// TIA Portal V17 export
// export: Created 2025-08-05T09:36:02.3274089Z, ExportSetting WithDefaults, DisplayName Totally Integrated Automation Portal, DisplayVersion V17, DisplayName TIA Portal Openness, DisplayVersion V17, DisplayName TIA Portal Version Control Interface, DisplayVersion V17, DisplayName SINAMICS Startdrive Advanced, DisplayVersion V17, DisplayName SINAMICS Startdrive G130, G150, S120, S150, SINAMICS MV, S210, DisplayVersion V17, DisplayName SINAMICS Startdrive G110M, G120, G120C, G120D, G120P, G115D, DisplayVersion V17, DisplayName STEP 7 Professional, DisplayVersion V17, DisplayName STEP 7 Safety, DisplayVersion V17, DisplayName WinCC Advanced, DisplayVersion V17
TYPE "typeSmcChillerHrle90a40cmIo"
// stored: IsFailsafeCompliant false
   STRUCT
      in { ExternalAccessible := 'False'; ExternalVisible := 'False'; ExternalWritable := 'False'} : Struct   // Lesen / Read
         fluidDischargeTempCH1 { ExternalAccessible := 'False'; ExternalVisible := 'False'; ExternalWritable := 'False'} : Real;   // Austrittstemperatur der zirkulierenden Flüssigkeit Kanal 1 / Outlet temperature of the circulating fluid channel 1
         fluidDischargeTempCH2 { ExternalAccessible := 'False'; ExternalVisible := 'False'; ExternalWritable := 'False'} : Real;   // Austrittstemperatur der zirkulierenden Flüssigkeit Kanal 2 / Outlet temperature of the circulating fluid channel 2
         reserve1 { ExternalAccessible := 'False'; ExternalVisible := 'False'; ExternalWritable := 'False'} : Word;   // Reserve
         reserve2 { ExternalAccessible := 'False'; ExternalVisible := 'False'; ExternalWritable := 'False'} : Word;   // Reserve
         fluidDischargePressureCH1 { ExternalAccessible := 'False'; ExternalVisible := 'False'; ExternalWritable := 'False'} : Real;   // Förderdruck der zirkulierenden Flüssigkeit Kanal 1 / Delivery pressure of the circulating fluid channel 1
         reserve3 { ExternalAccessible := 'False'; ExternalVisible := 'False'; ExternalWritable := 'False'} : Word;   // Reserve
         reserve4 { ExternalAccessible := 'False'; ExternalVisible := 'False'; ExternalWritable := 'False'} : Word;   // Reserve
         reserve5 { ExternalAccessible := 'False'; ExternalVisible := 'False'; ExternalWritable := 'False'} : Word;   // Reserve
         dataDisplay1 { ExternalAccessible := 'False'; ExternalVisible := 'False'; ExternalWritable := 'False'} : Real;   // Datenanzeige 1 / Data display 1
         dataDisplay2 { ExternalAccessible := 'False'; ExternalVisible := 'False'; ExternalWritable := 'False'} : Real;   // Datenanzeige 2 / Data display 2
         statusFlags1 { ExternalAccessible := 'False'; ExternalVisible := 'False'; ExternalWritable := 'False'} : Array[0..15] of Bool;   // Statuskennzeichen 1 / Status identifier 1
         alarmFlags1 { ExternalAccessible := 'False'; ExternalVisible := 'False'; ExternalWritable := 'False'} : Array[0..15] of Bool;   // Alarmmerker 1 / Alarm flag 1
         alarmFlags2 { ExternalAccessible := 'False'; ExternalVisible := 'False'; ExternalWritable := 'False'} : Array[0..15] of Bool;   // Alarmmerker 2 / Alarm flag 2
         alarmFlags3 { ExternalAccessible := 'False'; ExternalVisible := 'False'; ExternalWritable := 'False'} : Array[0..15] of Bool;   // Alarmmerker 3 / Alarm flag 3
         alarmFlags4 { ExternalAccessible := 'False'; ExternalVisible := 'False'; ExternalWritable := 'False'} : Array[0..15] of Bool;   // Alarmmerker 4 / Alarm flag 4
         alarmFlags5 { ExternalAccessible := 'False'; ExternalVisible := 'False'; ExternalWritable := 'False'} : Array[0..15] of Bool;   // Alarmmerker 5 / Alarm flag 5
      END_STRUCT;
      inOut { ExternalAccessible := 'False'; ExternalVisible := 'False'; ExternalWritable := 'False'} : Struct   // Lesen/Schreiben / Read/write
         fluidSetTempCH1 { ExternalAccessible := 'False'; ExternalVisible := 'False'; ExternalWritable := 'False'} : Real;   // Solltemperatur der zirkulierenden Flüssigkeit / Target temperature of the circulating fluid
         fluidSetTempCH2 { ExternalAccessible := 'False'; ExternalVisible := 'False'; ExternalWritable := 'False'} : Real;   // Umwälzflüssigkeitssolltemperatur als Offset von Kanal 1 (Sollwert Kanal 2 = Sollwert Kanal 1 + Offset Kanal 2) / Circulating fluid target temperature as offset for channel 1 (target value channel 2 = target value channel 1 + offset channel 2)
         controlBits { ExternalAccessible := 'False'; ExternalVisible := 'False'; ExternalWritable := 'False'} : Array[0..15] of Bool;   // Steuerbits / Control bits
         dataInstr { ExternalAccessible := 'False'; ExternalVisible := 'False'; ExternalWritable := 'False'} : Array[0..1] of Byte;   // Datenanweisungen / Data instructions
      END_STRUCT;
   END_STRUCT;
   // // in.statusFlags1[0] : Laufstatus / Running status
   // // in.statusFlags1[1] : Betriebsstoppalarm ausgelöst Status / Stop operation alarm triggered status
   // // in.statusFlags1[2] : Betriebsfortsetzungsalarm ausgelöst / Continue operation alarm triggered
   // // in.statusFlags1[3] : Reserve
   // // in.statusFlags1[4] : Abschluss der Vorbereitung (TEMP READY) Status / End of preparation (TEMP READY) status
   // // in.statusFlags1[5] : Reserve
   // // in.statusFlags1[6] : Reserve
   // // in.statusFlags1[7] : Reserve
   // // in.statusFlags1[8] : Reserve
   // // in.statusFlags1[9] : Reserve
   // // in.statusFlags1[10] : Reserve
   // // in.statusFlags1[11] : Reserve
   // // in.statusFlags1[12] : Reserve
   // // in.statusFlags1[13] : Reserve
   // // in.statusFlags1[14] : Reserve
   // // in.statusFlags1[15] : Gefrierschutzstatus / Freeze protection status
   // // in.alarmFlags1[0] : Niedriger Flüssigkeitsstand im Tank / Low fluid level in the tank
   // // in.alarmFlags1[1] : CH1 abnorm hohe Temperatur der zirkulierenden Flüssigkeit / CH1 abnormally high temperature of the circulating fluid
   // // in.alarmFlags1[2] : Reserve
   // // in.alarmFlags1[3] : Reserve
   // // in.alarmFlags1[4] : Ungewöhnlich hohe Rücklauftemperatur der zirkulierenden Flüssigkeit / Unusually high return temperature of the circulating fluid
   // // in.alarmFlags1[5] : Ungewöhnlich hoher Auslassdruck der zirkulierenden Flüssigkeit / Unusually high outlet pressure of the circulating fluid
   // // in.alarmFlags1[6] : Reserve
   // // in.alarmFlags1[7] : Hoher Druckanstieg der zirkulierenden Flüssigkeit / High pressure increase of the circulating fluid
   // // in.alarmFlags1[8] : Hoher Druckabfall der zirkulierenden Flüssigkeit / High pressure of the circulating fluid
   // // in.alarmFlags1[9] : Reserve
   // // in.alarmFlags1[10] : Ungewöhnlich niedrige Ansaugtemperatur des Kompressors / Unusually low intake temperature of the compressor
   // // in.alarmFlags1[11] : Reserve
   // // in.alarmFlags1[12] : Unnormaler Anstieg des Drucks im Kältemittelkreislauf (Hochdruckseite) / Abnormal pressure rise in the coolant circuit (high pressure side)
   // // in.alarmFlags1[13] : Reserve
   // // in.alarmFlags1[14] : Kältemittelleck / Coolant leak
   // // in.alarmFlags1[15] : Ungewöhnlicher Anstieg des Drucks im Kältemittelkreislauf (Niederdrucksei / Unusual pressure rise in the coolant circuit (low pressure side)
   // // in.alarmFlags2[0] : Ungewöhnlicher Druckabfall im Kältemittelkreislauf (Niederdruckseite) / Unusual pressure drop in the coolant circuit (low pressure side)
   // // in.alarmFlags2[1] : Kompressor läuft nicht / Compressor not running
   // // in.alarmFlags2[2] : Kommunikationsfehler / Communication error
   // // in.alarmFlags2[3] : Reserve
   // // in.alarmFlags2[4] : Reserve
   // // in.alarmFlags2[5] : Ausfall des Temperatursensors für den Auslass der CH1-Umlaufflüssigkeit（PT1) / Failure of the temperature sensor for the outlet of the CH1 circulation fluid （PT1)
   // // in.alarmFlags2[6] : Ausfall des Rücklauftemperatursensors der zirkulierenden Flüssigkeit（PT2) / Failure of the circulating fluid return temperature sensor （PT2)
   // // in.alarmFlags2[7] : Verdichter-Saugtemperatursensor defekt（TH2) / Compressor intake temperature sensor defective（TH2)
   // // in.alarmFlags2[8] : Ausfall des Drucksensors für die zirkulierende Flüssigkeit （PS1） / Failure of the pressure sensor for the circulating fluid （PS1）
   // // in.alarmFlags2[9] : Drucksensor des Kältemittelkreislaufs (Hochdruckseite) defekt（PS2） / Pressure sensor of the coolant circuit (high pressure side) defective（PS2）
   // // in.alarmFlags2[10] : Drucksensor des Kältemittelkreislaufs (Niederdruckseite) defekt（PS3） / Pressure sensor of the coolant circuit (low pressure side) defective（PS3）
   // // in.alarmFlags2[11] : Reserve
   // // in.alarmFlags2[12] : Reserve
   // // in.alarmFlags2[13] : Reserve
   // // in.alarmFlags2[14] : Kontakteingang 1 Signalerkennung / Contact input 1 signal detection
   // // in.alarmFlags2[15] : Kontakteingang 2 Signalerkennung / Contact input 2 signal detection
   // // in.alarmFlags3[0] : Reserve
   // // in.alarmFlags3[1] : Anstieg der elektrischen Leitfähigkeit / Increase in electrical conductivity
   // // in.alarmFlags3[2] : Rückgang der elektrischen Leitfähigkeit / Decrease in electrical conductivity
   // // in.alarmFlags3[3] : Ausfall des elektrischen Leitfähigkeitssensors / Failure of the electrical conductivity sensor
   // // in.alarmFlags3[4] : Ausfall des Verdichter-Drucktemperatursensors （TH1) / Failure of the compressor pressure and temperature sensor （TH1)
   // // in.alarmFlags3[5] : Anstieg der Verdichter-Austrittstemperatur / Increase in compressor outlet temperature
   // // in.alarmFlags3[6] : Reserve
   // // in.alarmFlags3[7] : Reserve
   // // in.alarmFlags3[8] : Reserve
   // // in.alarmFlags3[9] : Reserve
   // // in.alarmFlags3[10] : Ausfall des Ventilators / Failure of the ventilator
   // // in.alarmFlags3[11] : Reserve
   // // in.alarmFlags3[12] : Reserve
   // // in.alarmFlags3[13] : Verdichter-Wechselrichter-Fehler / Compressor inverter error
   // // in.alarmFlags3[14] : Störung des Pumpenbetriebs / Pump operation fault
   // // in.alarmFlags3[15] : Fehler im Pumpenumrichter / Error in the pump inverter
   // // in.alarmFlags4[0] : Reserve
   // // in.alarmFlags4[1] : CH2 abnormal hohe Temperatur der zirkulierenden Flüssig / CH2 abnormally high temperature of the circulating fluid
   // // in.alarmFlags4[2] : Ausfall des Temperatursensors für den Auslass der CH2-Umlaufflüssigkeit（PT3） / Failure of the temperature sensor for the outlet of the CH2 circulation fluid （PT3)
   // // in.alarmFlags4[3] : Speicherfehler 1 / Storage error 1
   // // in.alarmFlags4[4] : Speicherfehler 2 / Storage error 2
   // // in.alarmFlags4[5] : Reserve
   // // in.alarmFlags4[6] : Reserve
   // // in.alarmFlags4[7] : Abnormale Missing-Phase / Anti-Phase / Abnormal missing phase / anti-phase
   // // in.alarmFlags4[8] : Kommunikationsfehler des Verdichterwechselrichters / Communication error of the compressor inverter
   // // in.alarmFlags4[9] : Parameterfehler des Pumpenumrichters / Pump inverter parameter error
   // // in.alarmFlags4[10] : Kommunikationsfehler des Pumpenumrichters / Communication error of the pump inverter
   // // in.alarmFlags4[11] : Hinweis zur Wartung / Note on preventive maintenance
   // // in.alarmFlags4[12] : Kommunikationsfehler / Communication error
   // // in.alarmFlags4[13] : Interner Kommunikationsfehler / Internal communication error
   // // in.alarmFlags4[14] : Druckanstieg im Kältemittelkreislauf (Hochdruckseite) / Pressure rise in the coolant circuit (high pressure side)
   // // in.alarmFlags4[15] : Fehler in der Stromversorgung / Error in the power supply
   // // in.alarmFlags5[0] : Schalterbetätigung für den Druck im Kältemittelkreislauf (Hochdruckseite) / Switch actuation for the pressure in the coolant circuit (high pressure side)
   // // in.alarmFlags5[1] : Parameterfehler des Verdichterumrichters / Compressor inverter parameter error
   // // in.alarmFlags5[2] : Reserve
   // // in.alarmFlags5[3] : Reserve
   // // in.alarmFlags5[4] : Reserve
   // // in.alarmFlags5[5] : Reserve
   // // in.alarmFlags5[6] : Reserve
   // // in.alarmFlags5[7] : Reserve
   // // in.alarmFlags5[8] : Reserve
   // // in.alarmFlags5[9] : Reserve
   // // in.alarmFlags5[10] : Reserve
   // // in.alarmFlags5[11] : Reserve
   // // in.alarmFlags5[12] : Reserve
   // // in.alarmFlags5[13] : Reserve
   // // in.alarmFlags5[14] : Reserve
   // // in.alarmFlags5[15] : Reserve
   // // inOut.controlBits[0] : Befehl zum Starten der Operation / Command for starting the operation
   // // inOut.controlBits[1] : Flagge für Modusanforderung / Flag for mode request
   // // inOut.controlBits[2] : Alarm-Reset-Flag / Alarm reset flag
   // // inOut.controlBits[3] : Reserve
   // // inOut.controlBits[4] : Reserve
   // // inOut.controlBits[5] : Reserve
   // // inOut.controlBits[6] : Reserve
   // // inOut.controlBits[7] : Reserve
   // // inOut.controlBits[8] : Reserve
   // // inOut.controlBits[9] : Reserve
   // // inOut.controlBits[10] : Reserve
   // // inOut.controlBits[11] : Reserve
   // // inOut.controlBits[12] : Reserve
   // // inOut.controlBits[13] : Reserve
   // // inOut.controlBits[14] : Reserve
   // // inOut.controlBits[15] : Reserve
   // // inOut.dataInstr[0] : Datenanweisung 1 / Data instruction 1
   // // inOut.dataInstr[1] : Datenanweisung 2 / Data instruction 2
END_TYPE
